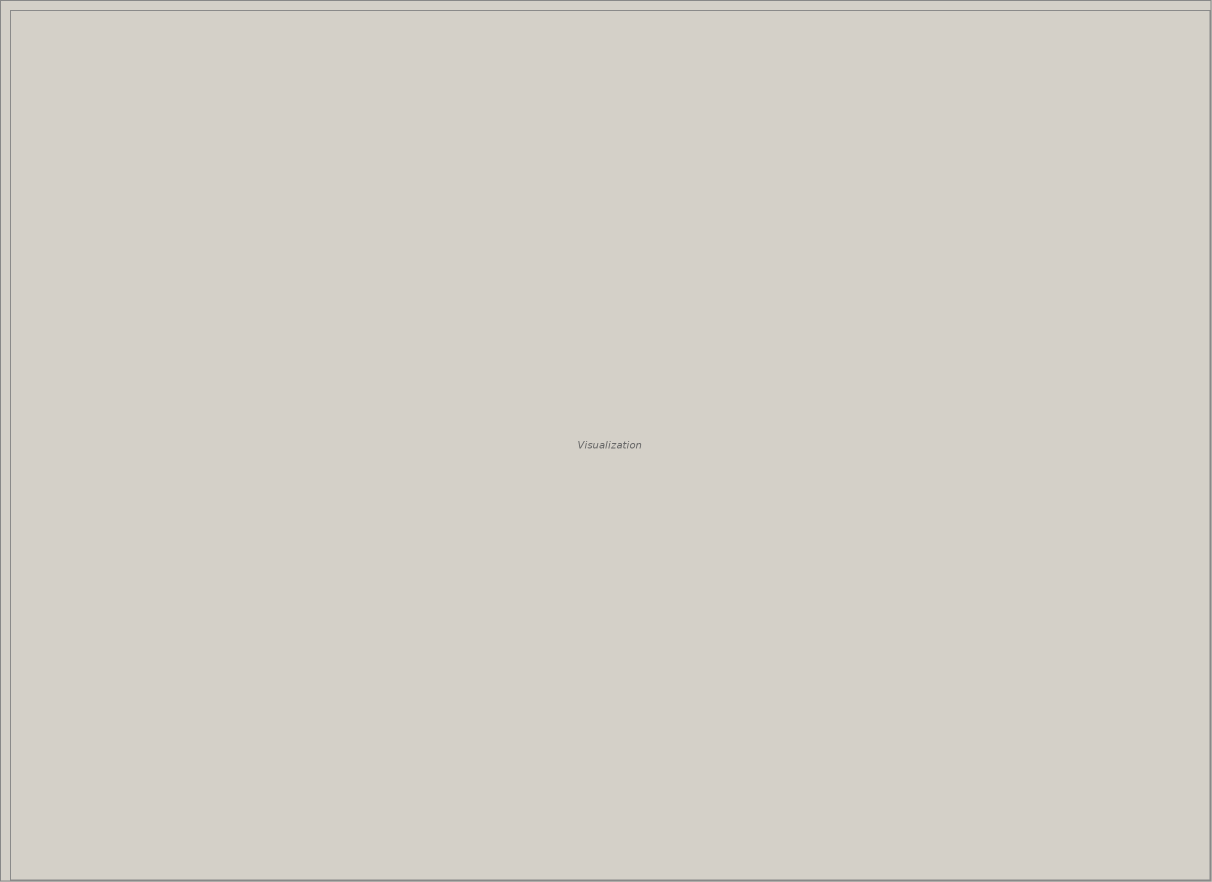
VISUALIZATION MAINVISU  // 1212x882
    TabControl (10,10 1200x870)
        shows Visualization()
        shows SlitSet()
        shows IO()
        [0]: TabTitle=Single Axis
        [1]: TabTitle=Slit Set
END_VISUALIZATION

(* stored: Version 1.1.0.1, ProductVersion 3.1.4020.12
   Visu MAINVISU: Id {0c75beb7-bbc6-400e-b853-9d5a64f7c839} *)
